Staubli VAL3: remMovAxis.pgx

program remMovAxis(string& sArgs[] (dimensions=1), string& sReturn[] (dimensions=1))
  local bool bOk
  local num nIndex
  local num nVal
  local string sAxis
  local string sVal
  local trsf trDest
begin
  // Move robot to a specific point along one axis,
  // keeping positions along other axes in the Cartesian
  // coordinate system static.
  //
  // Arguments are "AXIS NUMBER" e.g. "X 35"
  //
  logMsg("call remMovAxis")
  //parse args, expecting axis label and a number.
  //We already know we have exactly 2 args.
  nIndex=find(sArgs," ")
  sAxis=left(sArgs,nIndex)
  sVal=delete(sArgs,nIndex+1,0)
  toNum(sVal,nVal,bOk)
  if bOk
    call remCalcHere()
    trDest={nXHere,nYHere,nZHere,nRXHere,nRYHere,nRZHere}
    switch sAxis
      case "X"
        trDest.x=nVal
      break
      case "Y"
        trDest.y=nVal
      break
      case "Z"
        trDest.z=nVal
      break
      case "RX"
        trDest.rx=nVal
      break
      case "RY"
        trDest.ry=nVal
      break
      case "RZ"
        trDest.rz=nVal
      break
      default
        call remErrInvalid("MOVAXIS",sAxis,sReturn)
        return
      break
    endSwitch
    call remMovPoint(trDest,sReturn)
  else
    call remErrNum("MOVAXIS",sVal,sReturn)
  endIf
end
